// TwinCAT 3 PLC project TransportB
// ProgramVersion: 3.1.4023.0
// libraries:
//   Tc2_MC2, * (Beckhoff Automation GmbH)
//   Tc2_MC2_FlyingSaw, * (Beckhoff Automation GmbH)
//   Tc2_Standard, * (Beckhoff Automation GmbH)
//   Tc2_System, * (Beckhoff Automation GmbH)
//   Tc3_Module, * (Beckhoff Automation GmbH)
// project tree:
//   / PlcTask.TcTTO
//   POUs/ MAIN.TcPOU, Sensor.TcPOU, TransportSystemSlave.TcPOU
// (motion and I/O tree: see PLC project bohrmachine)
// real-time tasks:
//   TASK PlcTask: cycle T#10ms, priority 20, ADS port 350
//   TASK PlcTask1: cycle T#10ms, priority 21, ADS port 351
//   TASK PlcTask2: cycle T#10ms, priority 22, ADS port 352
//   TASK PlcTask3: cycle T#10ms, priority 23, ADS port 353
//   TASK ControllerTask: cycle T#10ms, priority 1, ADS port 354
//   TASK PlcTask4: cycle T#10ms, priority 24, ADS port 355
//   TASK PlcTask5: cycle T#10ms, priority 25, ADS port 356
// variable links:
//   TransportA/TransportA Instance <-> TransportB/TransportB Instance
//     PlcTask Outputs/MAIN.fbTransport.rActVelocity <-> PlcTask Inputs/MAIN.fbTransportSlave.rMasterVelocity
//   TransportB/TransportB Instance <-> NC-Task 1 SAF/Axes/TransportB
//     PlcTask Inputs/MAIN.fbTransportSlave.axisTransportB.NcToPlc <-> Outputs/ToPlc
//     PlcTask Outputs/MAIN.fbTransportSlave.axisTransportB.PlcToNc <-> Inputs/FromPlc
//   TransportB/TransportB Instance <-> Controller/Controller_Obj1 (ModuleController)
//     PlcTask Outputs/MAIN.fbTransportSlave.eZustand <-> TransportB/State
//     PlcTask Outputs/MAIN.fbTransportSlave.fbSensor.bWerkStueckLiegtAn <-> TransportB/WerkstueckLiegtAn
//     PlcTask Outputs/MAIN.fbTransportSlave.objID <-> InputIPointers/oidTransportB

CONFIGURATION TransportB
    RESOURCE PLC ON TwinCAT3
        TASK PlcTask(INTERVAL := T#10ms, PRIORITY := 22);
        PROGRAM MAIN WITH PlcTask : MAIN;
    END_RESOURCE
END_CONFIGURATION

// ---- POUs/MAIN.TcPOU
PROGRAM MAIN
VAR
	fbTransportSlave: TransportSystemSlave('MAIN.TPS_B');
END_VAR

fbTransportSlave();

{attribute 'call_after_init'}
METHOD Setup : BOOL
END_METHOD

END_PROGRAM

// ---- POUs/TransportSystemSlave.TcPOU
{attribute 'c++_compatible'}
FUNCTION_BLOCK TransportSystemSlave EXTENDS TcBaseModuleRegistered IMPLEMENTS I_TransportSlave
VAR_INPUT
END_VAR
VAR_OUTPUT
END_VAR
VAR
(*
Naive Implementierung um MC_GearInVelo / GearOut nachzubilden.
*)

	// ==== Motion Control ====
	axisTransportB: AXIS_REF;		// Slave
	fbMc_Power: MC_Power;			// Power
	fbMc_Halt: MC_Halt;				// Halt
	fbMc_MoveVelocity: MC_MoveVelocity; // continuous motion
	
	// ==== Inputs =====
	rMasterVelocity AT %I*: LREAL;	// Master velocity
	
	// ==== States ====
	eZustand AT %Q*: E_STATES_TRANSPORT_B := E_STATES_TRANSPORT_B.eHalted;	// aktueller Zustand
//	bReady: BOOL := FALSE;			// Achse bereit?

	// ==== Objects ====
	fbSensor: Sensor;
END_VAR

// ==== Inputs ====
axisTransportB.ReadStatus();

// ==== Object updates ====
fbSensor();

// ==== Statemachine ====
CASE eZustand OF
	E_STATES_TRANSPORT_B.eHalting:
		THIS^.Halting();

	E_STATES_TRANSPORT_B.eHalted:
		// idle

	E_STATES_TRANSPORT_B.eSyncing:
		THIS^.Syncing();

	E_STATES_TRANSPORT_B.eSynced:
		// idle
END_CASE

METHOD FB_reinit : BOOL
VAR_INPUT
END_VAR
SUPER^.FB_reinit();
END_METHOD

{attribute 'TcTypeSystem'}
{attribute 'no-analysis'}
{attribute 'c++_compatible'}
{attribute 'minimal_input_size' := '4'}
{attribute 'pack_mode' := '4'}
(* Anhalten *)
METHOD Halt : HRESULT
CASE eZustand OF
	E_STATES_TRANSPORT_B.EHALTED:
		Halt := S_OK;
		
	E_STATES_TRANSPORT_B.EHALTING:
		Halt := S_PENDING;
		
	ELSE
		THIS^.eZustand := E_STATES_TRANSPORT_B.eHalting;
		Halt := S_PENDING;
END_CASE
END_METHOD

METHOD PRIVATE Halting : BOOL
VAR_INPUT
END_VAR
fbMc_MoveVelocity(
	Axis := axisTransportB,
	Execute := FALSE
);

fbMc_Halt(
	Axis := axisTransportB,
	Execute := TRUE
);

IF fbMc_Halt.Done THEN
	fbMc_Halt(
		Axis := axisTransportB,
		Execute := FALSE
	);
	//bReady := FALSE;
	THIS^.eZustand := E_STATES_TRANSPORT_B.eHalted;
END_IF
END_METHOD

METHOD PRIVATE Syncing : BOOL
VAR_INPUT
END_VAR
// Achse starten und wenn Sie bereit ist, auf Master-Geschwindigkeit ziehen
// MC_POWER -> MC_MoveVelocity

// TODO jeden Baustein auf Fehler prüfen, evtl allgemeinen Zustand Error einführen

// Achse ist nicht bereit (nicht mit MC_Power freigegeben)
IF NOT fbMc_Power.Status THEN
	fbMc_Power(
		Axis := axisTransportB,
		Enable := TRUE,
		Enable_Positive := TRUE
	);
//	fbMc_MoveVelocity(
//		Execute := FALSE,
//		Axis := axisTransportB
//	);
ELSE // Achse ist bereit und beschleunigt auf Zielgeschwindigkeit
	fbMc_MoveVelocity(
		Execute := TRUE,
		Axis := axisTransportB,
		Direction := MC_Direction.MC_Positive_Direction,
		Velocity := rMasterVelocity
	);

	// Achse hat Zielgeschwindigkeit erreicht => Zustand: Synced
	IF fbMc_MoveVelocity.InVelocity THEN
		fbSensor.Reset();
		THIS^.eZustand := E_STATES_TRANSPORT_B.eSynced;
	END_IF	
END_IF
END_METHOD

{attribute 'TcTypeSystem'}
{attribute 'no-analysis'}
{attribute 'c++_compatible'}
{attribute 'minimal_input_size' := '4'}
{attribute 'pack_mode' := '4'}
(* Passe dich der Master-Geschwindigkeit an *)
METHOD SyncWithMaster : HRESULT
CASE eZustand OF
	E_STATES_TRANSPORT_B.ESYNCED:
		SyncWithMaster := S_OK;
		
	E_STATES_TRANSPORT_B.ESYNCING:
		SyncWithMaster := S_PENDING;
	
	ELSE
		THIS^.eZustand := E_STATES_TRANSPORT_B.eSyncing;
		SyncWithMaster := S_PENDING;	
END_CASE
END_METHOD

{attribute 'TcTypeSystem'}
{attribute 'no-analysis'}
{attribute 'c++_compatible'}
{attribute 'minimal_input_size' := '4'}
{attribute 'pack_mode' := '4'}
METHOD TcQueryInterface : HRESULT
VAR_INPUT
	iid	: REFERENCE TO IID;
	pipItf	: POINTER TO PVOID;
END_VAR
VAR
	ipTPS: I_TransportSlave;
END_VAR
IF GuidsEqual(ADR(iid), ADR(TC_GLOBAL_IID_LIST.IID_I_TransportSlave)) THEN
	ipTPS := THIS^;
	pipItf^ := ITCUNKNOWN_TO_PVOID(ipTPS);
	TcAddRef();
	TcQueryInterface := S_OK;
ELSE
	TcQueryInterface := SUPER^.TcQueryInterface(iid, pipItf);
END_IF
END_METHOD

END_FUNCTION_BLOCK

// ---- POUs/Sensor.TcPOU
FUNCTION_BLOCK Sensor
VAR_INPUT
END_VAR
VAR_OUTPUT
END_VAR
VAR
	bWerkStueckLiegtAn AT %Q*: BOOL := FALSE;
	fbTimer: TON;
	bTimerOn: BOOL := FALSE;
END_VAR

fbTimer(IN := bTimerOn, PT := T#5S);
IF fbTimer.Q THEN
	bWerkStueckLiegtAn := TRUE;
	bTimerOn := FALSE;
END_IF

METHOD PUBLIC Reset : BOOL
VAR_INPUT
END_VAR
bWerkStueckLiegtAn := FALSE;
bTimerOn := TRUE;
END_METHOD

END_FUNCTION_BLOCK
